# EPICS StreamDevice protocol: FW102_IOC/protocols/FW102.protocol
Terminator = CR;

resetPosition
{
	out "RESET %i";
	in "OK";
}

getPosition
{
	out "POS";
	in "%i";
}

setPosition
{
	out "SET %i";
	in "OK";
}

stop
{
	out "STOP";
	in "OK";
}
